(* IEC 61131-3 sources: volt/packages/volt-lsp-iec/test-corpus/pro2193/Device/Plc Logic/Application/09 Misc/Library Manager/FloatingPointUtils, 44 files *)

(* ---- ESPECIAL_FP_VALUE.dut ---- *)
TYPE ESPECIAL_FP_VALUE :
(
	NAN := 0,
	POSINF := 1,
	NEGINF := 2,
	EPS := 3,
	MAXVAL := 4,
	MINVAL := 5
);
END_TYPE

(* ---- GVL.gvl ---- *)
VAR_GLOBAL
	EXP_MASK_REAL : UDINT := 16#7F800000;
	EXP_OFFSET_REAL : INT := 23;
	MANT_MASK_REAL : UDINT := 16#7FFFFF;
	RES_EXP_REAL : UINT := 16#FF;
	EXP_BIAS_REAL : INT := 127;
	NORM_MANT_REAL : UDINT := 16#800000;
	MAX_MANT_REAL : UDINT := 16#FFFFFF;
	MIN_EXP_REAL : INT := (INT#1 - (EXP_BIAS_REAL + EXP_OFFSET_REAL));
	MAX_EXP_REAL : INT := (UINT_TO_INT(RES_EXP_REAL) - ((INT#1 + EXP_BIAS_REAL) + EXP_OFFSET_REAL));
	EXP_MASK_LREAL : ULINT := 16#7FF0000000000000;
	EXP_OFFSET_LREAL : INT := 52;
	MANT_MASK_LREAL : ULINT := 16#FFFFFFFFFFFFF;
	RES_EXP_LREAL : UINT := 16#7FF;
	EXP_BIAS_LREAL : INT := 1023;
	NORM_MANT_LREAL : ULINT := 16#10000000000000;
	MAX_MANT_LREAL : ULINT := 16#1FFFFFFFFFFFFF;
	MIN_EXP_LREAL : INT := (INT#1 - (EXP_BIAS_LREAL + EXP_OFFSET_LREAL));
	MAX_EXP_LREAL : INT := (UINT_TO_INT(RES_EXP_LREAL) - ((INT#1 + EXP_BIAS_LREAL) + EXP_OFFSET_LREAL));
	STR_NAN : STRING(16) := 'NaN';
	STR_PINF : STRING(16) := '+Inf';
	STR_NINF : STRING(16) := '-Inf';
	LINT_MAX : LINT := 16#7FFFFFFFFFFFFFFF;
	INT_MAX : INT := 16#7FFF;
	INT_MIN : INT := -16#8000;
	DINT_MIN : DINT := -16#8000000;
	DINT_MAX : DINT := 16#7FFFFFFF;
END_VAR

(* ---- CEIL.pou ---- *)
FUNCTION CEIL : LREAL
VAR_INPUT
	F : LREAL;
END_VAR
END_FUNCTION

(* ---- CEILF.pou ---- *)
FUNCTION CEILF : REAL
VAR_INPUT
	F : REAL;
END_VAR
END_FUNCTION

(* ---- CHAREQCI.pou ---- *)
FUNCTION CHAREQCI : BOOL
VAR_INPUT
	C1 : BYTE;
	C2 : BYTE;
END_VAR
END_FUNCTION

(* ---- COMPOSELREAL.pou ---- *)
FUNCTION COMPOSELREAL : BOOL
VAR_INPUT
	LIM : LINT;
	IE : INT;
END_VAR
VAR_OUTPUT
	F : LREAL;
END_VAR
END_FUNCTION

(* ---- COMPOSELREALRAW.pou ---- *)
FUNCTION COMPOSELREALRAW : LREAL
VAR_INPUT
	BS : BOOL;
	UIE : UINT;
	ULIM : ULINT;
END_VAR
END_FUNCTION

(* ---- COMPOSEREAL.pou ---- *)
FUNCTION COMPOSEREAL : BOOL
VAR_INPUT
	DIM : DINT;
	IE : INT;
END_VAR
VAR_OUTPUT
	F : REAL;
END_VAR
END_FUNCTION

(* ---- COMPOSEREALRAW.pou ---- *)
FUNCTION COMPOSEREALRAW : REAL
VAR_INPUT
	BS : BOOL;
	UIE : UINT;
	UDIM : UDINT;
END_VAR
END_FUNCTION

(* ---- DESERIALIZEHEXREAL.pou ---- *)
FUNCTION DESERIALIZEHEXREAL : BOOL
VAR_INPUT
	PS : POINTER TO BYTE;
END_VAR
VAR_OUTPUT
	LIM : LINT;
	IE : INT;
	XNAN : BOOL;
	XINF : BOOL;
END_VAR
END_FUNCTION

(* ---- EXTRACTLREAL.pou ---- *)
FUNCTION EXTRACTLREAL : BOOL
VAR_INPUT
	F : LREAL;
END_VAR
VAR_OUTPUT
	IE : INT;
	LIM : LINT;
	XNAN : BOOL;
	XINF : BOOL;
END_VAR
END_FUNCTION

(* ---- EXTRACTLREALRAW.pou ---- *)
FUNCTION EXTRACTLREALRAW : BOOL
VAR_INPUT
	F : LREAL;
END_VAR
VAR_OUTPUT
	BS : BOOL;
	UIE : UINT;
	ULIM : ULINT;
END_VAR
END_FUNCTION

(* ---- EXTRACTREAL.pou ---- *)
FUNCTION EXTRACTREAL : BOOL
VAR_INPUT
	F : REAL;
END_VAR
VAR_OUTPUT
	IE : INT;
	DIM : DINT;
	XNAN : BOOL;
	XINF : BOOL;
END_VAR
END_FUNCTION

(* ---- EXTRACTREALRAW.pou ---- *)
FUNCTION EXTRACTREALRAW : BOOL
VAR_INPUT
	F : REAL;
END_VAR
VAR_OUTPUT
	BS : BOOL;
	UIE : UINT;
	UDIM : UDINT;
END_VAR
END_FUNCTION

(* ---- FLOOR.pou ---- *)
FUNCTION FLOOR : LREAL
VAR_INPUT
	F : LREAL;
END_VAR
END_FUNCTION

(* ---- FLOORF.pou ---- *)
FUNCTION FLOORF : REAL
VAR_INPUT
	F : REAL;
END_VAR
END_FUNCTION

(* ---- FLOORTEST.pou ---- *)
FUNCTION FLOORTEST : LREAL
VAR_INPUT
	F : LREAL;
END_VAR
END_FUNCTION

(* ---- GETLREALSPECIALVAL.pou ---- *)
FUNCTION GETLREALSPECIALVAL : LREAL
VAR_INPUT
	SV : ESpecial_FP_Value;
END_VAR
END_FUNCTION

(* ---- GETREALSPECIALVAL.pou ---- *)
FUNCTION GETREALSPECIALVAL : REAL
VAR_INPUT
	SV : ESpecial_FP_Value;
END_VAR
END_FUNCTION

(* ---- HEXDIGVAL.pou ---- *)
FUNCTION HEXDIGVAL : BYTE
VAR_INPUT
	C : BYTE;
END_VAR
END_FUNCTION

(* ---- HEXSTRTOLREAL.pou ---- *)
FUNCTION HEXSTRTOLREAL : BOOL
VAR_INPUT
	STR : STRING;
END_VAR
VAR_OUTPUT
	F : LREAL;
END_VAR
END_FUNCTION

(* ---- HEXSTRTOREAL.pou ---- *)
FUNCTION HEXSTRTOREAL : BOOL
VAR_INPUT
	STR : STRING;
END_VAR
VAR_OUTPUT
	F : REAL;
END_VAR
END_FUNCTION

(* ---- INSERTSTR.pou ---- *)
FUNCTION INSERTSTR : INT
VAR_INPUT
	PDST : POINTER TO BYTE;
	ISTARTINDEX : INT;
	PSRC : POINTER TO BYTE;
END_VAR
END_FUNCTION

(* ---- ISHEXDIG.pou ---- *)
FUNCTION ISHEXDIG : BOOL
VAR_INPUT
	C : BYTE;
END_VAR
END_FUNCTION

(* ---- ISLREALNAN.pou ---- *)
FUNCTION ISLREALNAN : BOOL
VAR_INPUT
	F : LREAL;
END_VAR
END_FUNCTION

(* ---- ISLREALNEGINFINITY.pou ---- *)
FUNCTION ISLREALNEGINFINITY : BOOL
VAR_INPUT
	F : LREAL;
END_VAR
END_FUNCTION

(* ---- ISLREALNUMBER.pou ---- *)
FUNCTION ISLREALNUMBER : BOOL
VAR_INPUT
	F : LREAL;
END_VAR
END_FUNCTION

(* ---- ISLREALPOSINFINITY.pou ---- *)
FUNCTION ISLREALPOSINFINITY : BOOL
VAR_INPUT
	F : LREAL;
END_VAR
END_FUNCTION

(* ---- ISREALNAN.pou ---- *)
FUNCTION ISREALNAN : BOOL
VAR_INPUT
	F : REAL;
END_VAR
END_FUNCTION

(* ---- ISREALNEGINFINITY.pou ---- *)
FUNCTION ISREALNEGINFINITY : BOOL
VAR_INPUT
	F : REAL;
END_VAR
END_FUNCTION

(* ---- ISREALNUMBER.pou ---- *)
FUNCTION ISREALNUMBER : BOOL
VAR_INPUT
	F : REAL;
END_VAR
END_FUNCTION

(* ---- ISREALPOSINFINITY.pou ---- *)
FUNCTION ISREALPOSINFINITY : BOOL
VAR_INPUT
	F : REAL;
END_VAR
END_FUNCTION

(* ---- LREALTOHEXSTR.pou ---- *)
FUNCTION LREALTOHEXSTR : STRING(32)
VAR_INPUT
	F : LREAL;
END_VAR
END_FUNCTION

(* ---- LREALTOSTR.pou ---- *)
FUNCTION LREALTOSTR : STRING(32)
VAR_INPUT
	F : LREAL;
END_VAR
END_FUNCTION

(* ---- REALTOHEXSTR.pou ---- *)
FUNCTION REALTOHEXSTR : STRING(32)
VAR_INPUT
	F : REAL;
END_VAR
END_FUNCTION

(* ---- REALTOSTR.pou ---- *)
FUNCTION REALTOSTR : STRING(16)
VAR_INPUT
	F : REAL;
END_VAR
END_FUNCTION

(* ---- SCANCONSTI.pou ---- *)
FUNCTION SCANCONSTI : BOOL
VAR_INPUT
	PS : POINTER TO BYTE;
	PSCONST : POINTER TO BYTE;
END_VAR
VAR_IN_OUT
	IDX : INT;
END_VAR
END_FUNCTION

(* ---- SCANHEXNUMERAL.pou ---- *)
FUNCTION SCANHEXNUMERAL : BOOL
VAR_INPUT
	PS : POINTER TO BYTE;
END_VAR
VAR_OUTPUT
	LI : LINT;
END_VAR
VAR_IN_OUT
	IDX : INT;
END_VAR
END_FUNCTION

(* ---- SERIALIZEHEXREAL.pou ---- *)
FUNCTION SERIALIZEHEXREAL : STRING(32)
VAR_INPUT
	LIM : LINT;
	IE : INT;
END_VAR
END_FUNCTION

(* ---- STRTOLREAL.pou ---- *)
FUNCTION STRTOLREAL : LREAL
VAR_INPUT
	STR : STRING;
END_VAR
END_FUNCTION

(* ---- STRTOREAL.pou ---- *)
FUNCTION STRTOREAL : REAL
VAR_INPUT
	STR : STRING;
END_VAR
END_FUNCTION

(* ---- TOHEXNUMERAL.pou ---- *)
FUNCTION TOHEXNUMERAL : INT
VAR_INPUT
	PDST : POINTER TO BYTE;
	LI : LINT;
END_VAR
END_FUNCTION

(* ---- TRUNCATE.pou ---- *)
FUNCTION TRUNCATE : LREAL
VAR_INPUT
	F : LREAL;
END_VAR
END_FUNCTION

(* ---- TRUNCATEF.pou ---- *)
FUNCTION TRUNCATEF : REAL
VAR_INPUT
	F : REAL;
END_VAR
END_FUNCTION
